// TIA Portal V18 export
TYPE "udt_Waypoint"
// stored: IsFailsafeCompliant false
   STRUCT
      baseAxis : Real;
      arm1Axis : Real;
      arm2Axis : Real;
      arm3Axis : Real;
      toolAxis : Real;
   END_STRUCT;
END_TYPE
